PROPERTY PickPlaceDataToPass : ST_PickPlace
GET
PickPlaceDataToPass := _PickPlaceDataToPass;
END_GET
END_PROPERTY

END_FUNCTION_BLOCK

// Machine/EquipmentModules/Functional Layer/FB_Robot_PrePlate
FUNCTION_BLOCK FB_Robot_PrePlate EXTENDS FB_Robot
VAR
    // Sub module definitions here

    Detail_SIM_TON : TON;
END_VAR

VAR

    Plates : ST_Plates;

END_VAR

METHOD CyclicLogic
VAR_INPUT
END_VAR

VAR

END_VAR
IF NOT _InitComplete THEN
    _InitComplete := Initialize();
    RETURN;
END_IF

SUPER^.CyclicLogic();

UI_MessageBox();
END_METHOD

METHOD CyclicLogicSimulation : BOOL
VAR_INPUT
END_VAR
END_METHOD

METHOD ExecuteDetail : BOOL
VAR_INPUT
    StepToRun : UDINT;
END_VAR
ExecuteDetail := FALSE;

CASE Handshake_Step OF
    0:
        Robot.Handshake.OUT.Execute_Step    := TRUE;
        Robot.Handshake.OUT.Execute_StepNum := UDINT_TO_UINT(StepToRun);

        IF Robot.Handshake.IN.Executing_Step = TRUE THEN
            Handshake_Step := 1;
        END_IF

    1:
        IF Robot.Handshake.IN.Executing_Step = FALSE AND Robot.Handshake.IN.StepComplete = TRUE THEN
            Handshake_Step := 2;
        END_IF

    2:
        Robot.Handshake.OUT.Execute_Step    := FALSE;
        Robot.Handshake.OUT.Execute_StepNum := 0;

        IF Robot.Handshake.IN.StepComplete = FALSE THEN
            ExecuteDetail  := TRUE;
            Handshake_Step := 0;
        END_IF

END_CASE
END_METHOD

METHOD PROTECTED ExecuteDetail_SIM : BOOL
VAR_INPUT
    StepToRun : UDINT;
END_VAR
IF WaitSync_Handler(E_WaitSync.PRESS_PREPLATE_SIM_SYNC) THEN
    ExecuteDetail_SIM := TRUE;
END_IF
END_METHOD

METHOD ExecuteStep : BOOL
VAR_INPUT
    Step : ST_CSV_Step;
END_VAR

VAR_INST
    LastExecutionTime  : ULINT; // 64-bit unsigned for F_GetSystemTime
    CurrentTime        : ULINT;
    LastHourCheck      : ULINT;
    ExecutionTime      : ULINT;
    NailPlateTimes     : ARRAY[0..9] OF ULINT; // Buffer for 10 samples
    TotalTime          : REAL; // Use REAL for floating-point calc
    TimeBufferIndex    : INT  := 0;
    TimeSampleCount    : INT  := 0;
    NailPlatesPerMin   : REAL := 0.0; // Plates per minute
    NailPlatesPerHour  : REAL := 0.0; // Plates per hour
    HourAccumulator    : REAL := 0.0;
    ShiftSampleCount   : INT  := 0;
    ShiftNailPlateAvgs : ARRAY[0..7] OF REAL; // 8-hour shift storage
    ShiftHourIndex     : INT := 0;
    BoardNumber        : INT;
END_VAR
ExecuteStep := FALSE;

CASE Step.seqName OF
    E_CommandName.BoardInfo:
        BoardNumber := STRING_TO_INT(Step.Details[1].Datas[2]);
		ExecuteStep := TRUE;
    E_CommandName.NailPlate:
        // Initialize timing on first run
        IF TimeSampleCount = 0 AND TimeBufferIndex = 0 AND ShiftSampleCount = 0 THEN
            LastExecutionTime := F_GetSystemTime();
            LastHourCheck     := LastExecutionTime;
        END_IF

        NailPlateParse(Step, Plates);

        // Clear out array first
        Robot.Clear_DataToSend();

        // First entry is always step type
        Robot.RecipeData_ToSend[0] := E_CommandName.NailPlate;

        Robot.RecipeData_ToSend[1] := UDINT_TO_DINT(Step.DetailCount);
        Robot.RecipeData_ToSend[2] := (Plates.Plates[DetailIndex].PlateNumber + (BoardNumber * 10));
        Robot.RecipeData_ToSend[3] := ExtractNumFromString(Plates.Plates[DetailIndex].PlateGauge);
        Robot.RecipeData_ToSend[4] := REAL_TO_DINT(Plates.Plates[DetailIndex].PlateWidth * 10);
        Robot.RecipeData_ToSend[5] := REAL_TO_DINT(Plates.Plates[DetailIndex].PlateHeight * 10);
        Robot.RecipeData_ToSend[6] := REAL_TO_DINT(Plates.Plates[DetailIndex].PlatePlaceY * 10);
        Robot.RecipeData_ToSend[7] := REAL_TO_DINT(Plates.Plates[DetailIndex].PlatePlaceAngle * 10);

        IF Plates.Plates[DetailIndex].TopOrBottom = 'Top' THEN
            Robot.RecipeData_ToSend[8] := 1;
        ELSIF Plates.Plates[DetailIndex].TopOrBottom = 'Bottom' THEN
            Robot.RecipeData_ToSend[8] := 2;
        ELSE
            Robot.RecipeData_ToSend[8] := 0;
        END_IF

        IF _InSimulation THEN
            IF ExecuteDetail_SIM(Step.seqID) THEN
                DetailIndex := DetailIndex + 1;
                Detail_SIM_TON(IN := FALSE);
            END_IF
        ELSE
            IF ExecuteDetail(Step.seqID) THEN
                CurrentTime   := F_GetSystemTime();
                ExecutionTime := CurrentTime - LastExecutionTime;

                // Convert 100ns units to seconds (100ns * 10,000,000 = 1s)
                NailPlateTimes[TimeBufferIndex] := ExecutionTime;
                TimeBufferIndex                 := TimeBufferIndex + 1;

                IF TimeBufferIndex >= 10 THEN
                    TimeBufferIndex := 0;
                END_IF

                IF TimeSampleCount < 10 THEN
                    TimeSampleCount := TimeSampleCount + 1;
                END_IF

                TotalTime := 0.0;

                FOR i := 0 TO TimeSampleCount - 1 DO
                    TotalTime := TotalTime + ULINT_TO_REAL(NailPlateTimes[i]) / 10000000.0; // Convert to seconds
                END_FOR

                IF TotalTime > 0.0 THEN
                    // Calculate plates per minute (samples per average time in seconds)
                    NailPlatesPerMin := (TimeSampleCount / TotalTime) * 60.0;
                    // Calculate plates per hour
                    NailPlatesPerHour := NailPlatesPerMin * 60.0;
                END_IF

                // Shift-long tracking
                HourAccumulator  := HourAccumulator + 1.0; // Count each plate
                ShiftSampleCount := ShiftSampleCount + 1;

                // Check if an hour has passed (36000000000 100ns units = 1 hour)
                IF (CurrentTime - LastHourCheck) >= 36000000000 THEN
                    IF ShiftSampleCount > 0 THEN
                        // Store hourly rate (plates per hour)
                        ShiftNailPlateAvgs[ShiftHourIndex] := (HourAccumulator * 3600.0) / (ULINT_TO_REAL(CurrentTime - LastHourCheck) / 10000000.0);
                        ShiftHourIndex                     := ShiftHourIndex + 1;
                        HourAccumulator                    := 0.0;
                        ShiftSampleCount                   := 0;
                    END_IF

                    LastHourCheck := CurrentTime;

                    IF ShiftHourIndex >= 8 THEN
                        ShiftHourIndex := 0; // Start new shift
                    END_IF
                END_IF

                LastExecutionTime := CurrentTime;
                DetailIndex       := DetailIndex + 1;
            END_IF
        END_IF

        IF DetailIndex > Step.DetailCount THEN
            DetailIndex := 1;
            ExecuteStep := TRUE;
        END_IF

ELSE
    ExecuteStep := TRUE;

END_CASE
END_METHOD

METHOD HMIControl
VAR_INPUT
END_VAR
END_METHOD

//! @summary Basic module initialization logic
METHOD PROTECTED Initialize : BOOL;
VAR
    i                        : UDINT;
    varInfo                  : __SYSTEM.VAR_INFO;
    AllSubUnitsInitialized   : BOOL := TRUE;
    AllComponentsInitialized : BOOL := TRUE;
END_VAR

//! @description This method is called by <c>CyclicLogic()</c> as required
Initialize := FALSE;

CASE DescendantSequenceState OF
    0:
        RegisterComponent(Robot);

        _LogModeChanges         := FALSE;
        _LogStateChanges        := FALSE;
        DescendantSequenceState := DescendantSequenceState + 10;

    10:
        //Setup Custom modes here

        (*CustomModes(eMode                          :=,
                    sName                          :=,
                    bDisableClearing               :=,
                    bDisableStarting               :=,
                    bDisableSuspended              :=,
                    bDisableStopping               :=,
                    bDisableAborting               :=,
                    bDisableHolding                :=,
                    bDisableHeld                   :=,
                    bDisableUnholding              :=,
                    bDisableSuspending             :=,
                    bDisableUnsuspending           :=,
                    bDisableResetting              :=,
                    bDisableIdle                   :=,
                    bDisableCompleting             :=,
                    bDisableComplete               :=,
                    bEnableUnitModeChangeStopped   :=,
                    bEnableUnitModeChangeIdle      :=,
                    bEnableUnitModeChangeSuspended :=,
                    bEnableUnitModeChangeExecute   :=,
                    bEnableUnitModeChangeAborted   :=,
                    bEnableUnitModeChangeHeld      :=,
                    bEnableUnitModeChangeComplete  :=,
                    bError                         =>,
                    nErrorId                       =>);*)

        DescendantSequenceState := DescendantSequenceState + 10;

    20:
        //Copy Mode names

        FOR i := 1 TO 3 DO
            ModeNames[i] := F_UnitModeToString(UDINT_TO_DINT(i));
        END_FOR

        RegisterExternalController(Controller := fbControlSourceHMI);
        fbControlSourceHMI.CyclicLogic();
        DescendantSequenceState := DescendantSequenceState + 10;

    30:
        //Call the Super

        IF SUPER^.Initialize() THEN
            DescendantSequenceState := DescendantSequenceState + 10;
        END_IF

    40:
        Initialize := TRUE;
END_CASE
END_METHOD

METHOD UI_MessageBox : BOOL
VAR_INPUT
END_VAR

VAR
    result : USINT;
END_VAR
IF Robot.Handshake.IN.ErrorPresent THEN
    CASE Robot.Handshake.IN.MessageNumber OF

        //////////////////////////// PREPLATE ROBOT ERRORS ////////////////////////////
        0:

            // Idle State Should not have an error of 0

            ///////// 1-29 PROCESS ERRORS /////////
        1:
            // PrePlate ERROR_REPEATEDSTEP_R1

            result := RaiseMessageBox(Header   := 'Repeated Step Warning.',
                                      Message1 := 'Robot is trying to repeat last step',
                                      Message3 := 'Choose RETRY to retry check',
                                      Message4 := 'Choose ABORT to reset robot',
                                      Btn3     := 'Retry',
                                      Btn4     := 'Override',
                                      Btn5     := 'Abort',
                                      Severity := TcEventSeverity.Error);

        2:
            // PrePlate ERROR_STEP_NOT_FOUND

            result := RaiseMessageBox(Header   := 'Step Not Found Warning.',
                                      Message1 := 'Robot is trying execute a step that does not exist',
                                      Message2 := 'Choose RETRY to retry check',
                                      Message3 := 'Choose OVERRIDE to override warning',
                                      Message4 := 'Choose ABORT to reset robot',
                                      Btn3     := 'Retry',
                                      Btn4     := 'Override',
                                      Btn5     := 'Abort',
                                      Severity := TcEventSeverity.Error);

        3:
            // PrePlate ERROR_PROCESSING_DATA

            result := RaiseMessageBox(Header   := 'Processing Data Error',
                                      Message1 := 'Check robot log for more information',
                                      Message2 := 'Choose RETRY to retry data processing',
                                      Message3 := 'Choose ABORT to reset robot',
                                      Btn3     := 'RETRY',
                                      Btn5     := 'ABORT',
                                      Severity := TcEventSeverity.Error);

        4:
            // PrePlate ERROR_NORUNUNIT

            result := RaiseMessageBox(Header   := 'IO Device not Connected.',
                                      Message1 := 'Check error log for more details',
                                      Message3 := 'click OK when ready to continue',
                                      Btn5     := 'OK',
                                      Severity := TcEventSeverity.Error);

        5:
            // PrePlate ERROR_NO_DATA_FILE

            result := RaiseMessageBox(Header   := 'No Data File Found.',
                                      Message1 := 'Resend data to robot and choose RETRY',
                                      Message3 := 'Choose ABORT to start recovery process',
                                      Btn3     := 'RETRY',
                                      Btn5     := 'ABORT',
                                      Severity := TcEventSeverity.Error);

        6:
            // PrePlate ERROR_ABORT

            result := RaiseMessageBox(Header   := 'Abort Error',
                                      Message1 := 'Aborting',
                                      Message3 := 'Select ABORT to continue.',
                                      Btn3     := 'ABORT',
                                      Severity := TcEventSeverity.Error);

        10:
            // Press Error ERROR_ABORT (Left magnet handoff not extending)

            result := RaiseMessageBox(Header   := 'Left magnet handoff not extending',
                                      Message1 := 'Make sure air on and extend sensor is connected correctly ',
                                      Message3 := 'System will continue when extend signal is triggered',
                                      Btn3     := 'OVERRIDE',
                                      Severity := TcEventSeverity.Info);

        11:
            // Press Error ERROR_ABORT (Right magnet handoff not extending)

            result := RaiseMessageBox(Header   := 'Right magnet handoff not extending',
                                      Message1 := 'Make sure air on and extend sensor is connected correctly ',
                                      Message3 := 'System will continue when extend signal is triggered',
                                      Btn3     := 'OVERRIDE',
                                      Severity := TcEventSeverity.Info);

        30:
            // PrePlate Error ERROR_UNKNOWNERROR_R1

            result := RaiseMessageBox(Header   := 'Unknown Robot Error',
                                      Message1 := 'Check the pendant for additional information.',
                                      Message3 := 'Press OK to continue.',
                                      Btn5     := 'OK',
                                      Severity := TcEventSeverity.Error);

        31:
            // PrePlate ERROR_PLATEDROPPED_R1

            result := RaiseMessageBox(Header   := 'PrePlate Robot Dropped Plate.',
                                      Message1 := 'Robot no longer holding plate.',
                                      Message3 := 'Choose ABORT to reset robot',
                                      Btn2     := 'Discard',
                                      Btn3     := 'Re-Pick',
                                      Btn4     := 'Override',
                                      Btn5     := 'Abort',
                                      Severity := TcEventSeverity.Error);

        32:
            // PrePlate ERROR_TWO_PLATES_DROPPED

            result := RaiseMessageBox(Header   := 'PrePlate Robot Dropped Plate Twice.',
                                      Message1 := 'Check End Of Arm Tool',
                                      Message3 := 'Choose OVERRIDE if nothing wrong',
                                      Message4 := 'Choose ABORT to reset robot',
                                      Btn2     := 'Discard',
                                      Btn3     := 'Re-Pick',
                                      Btn4     := 'Override',
                                      Btn5     := 'Abort',
                                      Severity := TcEventSeverity.Error);

        33:
            // Press ERROR_NO_MORE_MAGS

            // This one includes dynamic text for plate size

            // We'll place that dynamic content in one message for clarity

            result := RaiseMessageBox(Header   := 'No more magazines.',
                                      Message1 := CONCAT('Plate size = ', Plates.Plates[DetailIndex].PlateDimensions),
                                      Message2 := CONCAT('Plate gauge = ', Plates.Plates[DetailIndex].PlateGauge),
                                      Message3 := 'click OK when magazines are filled',
                                      Btn3     := 'Skip',
                                      Btn5     := 'OK',
                                      Severity := TcEventSeverity.Error);

        34:
            // PrePlate ERROR_EOAT_EXT_FAILURE

            result := RaiseMessageBox(Header   := 'EOAT Failed to Extend.',
                                      Message1 := 'Check EOAT for any blockage',
                                      Message2 := 'Choose DISABLE to disable check',
                                      Message3 := 'Choose RETRY to retry check',
                                      Message4 := 'Choose OVERRIDE to override warning',
                                      Message5 := 'Choose ABORT to reset robot',
                                      Btn2     := 'Disable',
                                      Btn3     := 'Retry',
                                      Btn4     := 'Override',
                                      Btn5     := 'Abort',
                                      Severity := TcEventSeverity.Error);

        35:
            // PrePlate ERROR_PLATE_NOT_FOUND

            result := RaiseMessageBox(Header   := 'Specified Plate does not Exist.',
                                      Message1 := 'Check data',
                                      Message2 := 'Choose RETRY to retry check',
                                      Message3 := 'Choose OVERRIDE to override warning',
                                      Message4 := 'Choose ABORT to reset robot',
                                      Btn3     := 'Retry',
                                      Btn4     := 'Override',
                                      Btn5     := 'Abort',
                                      Severity := TcEventSeverity.Error);

        36:
            // PrePlate ERROR_PLACE_OUT_OF_REACH

            result := RaiseMessageBox(Header   := 'Robot Out of Reach',
                                      Message1 := 'Check data',
                                      Message3 := 'Choose DISCARD to discard plate and move on to next one.',
                                      Btn3     := 'DISCARD',
                                      Btn5     := 'RECOVER',
                                      Severity := TcEventSeverity.Error);

        37:
            // PrePlate ERROR_UNRECOGNIZED_WORLD_ZONE

            result := RaiseMessageBox(Header   := 'Robot Unrecognized Position.',
                                      Message1 := 'Jog Robot to safe position and retry move home',
                                      Btn5     := 'RETRY',
                                      Severity := TcEventSeverity.Error);

        38:
            // PrePlate ERROR_PRESS_TASK_STOPPED

            result := RaiseMessageBox(Header   := 'Press Task Stopped.',
                                      Message1 := 'Make sure all tasks are enabled on the robot.',
                                      Btn5     := 'Retry',
                                      Severity := TcEventSeverity.Error);

        40:
            // PrePlate ERROR_NO_HANDSHAKE_ROBOT

            result := RaiseMessageBox(Header   := 'Robot - Waiting to Handshake',
                                      Message1 := 'The PLC and robot may be out of sync',
                                      Btn5     := 'Retry',
                                      Severity := TcEventSeverity.Error);

        41:
            // PrePlate ERROR_BAD_BOARD_DATA

            result := RaiseMessageBox(Header   := 'Bad Board Data',
                                      Message1 := 'Preplate CSV board data has boards that are too long/short/thick to be ran',
                                      Message3 := 'Check files and upload new files when fixed',
                                      Severity := TcEventSeverity.Error);

        42:
            // PrePlate ERROR_BAD_NAIL_DATA

            result := RaiseMessageBox(Header   := 'Bad Nail Plate Data',
                                      Message1 := 'Preplate CSV nail plate data has incorrect plate sizes',
                                      Message3 := 'Check files and upload new files when fixed',
                                      Severity := TcEventSeverity.Error);

        43:
            // PrePlate ERROR_FAILED_TO_PLACE

            result := RaiseMessageBox(Header   := 'PP Robot Failed to Place Nail Plate',
                                      Message1 := 'PrePlate robot still holding a nail plate after attempting to place it',
                                      Message3 := 'Select RETRY to have robot attempt to place nail plate again',
                                      Btn3     := 'Retry',
                                      Severity := TcEventSeverity.Error);

        44:
            // PrePlate ERROR_MAG_IN_DIS_RACK

            result := RaiseMessageBox(Header   := 'Only Available Magazine is in a Disabled Rack',
                                      Message1 := 'Re-Enable Rack',
                                      Message3 := 'Choose RETRY to attempt Finding Valid Mgazine',
                                      Btn5     := 'Retry',
                                      Severity := TcEventSeverity.Error);

        45:
            // PrePlate error nail plate skipped

            // Also includes dynamic text for plate size

            result := RaiseMessageBox(Header   := 'Nail plate Skipped',
                                      Message1 := 'Nail plate not available',
                                      Message3 := CONCAT('Nail plate size: ', Plates.Plates[DetailIndex].PlateDimensions),
                                      Btn5     := 'OK',
                                      Severity := TcEventSeverity.Error);

        50:
            result := RaiseMessageBox(Header   := 'Robot Read Bad Board Data',
                                      Message1 := 'Preplate CSV board data has boards that are too long/short/thick to be ran',
                                      Message3 := 'Check files and upload new files when fixed',
                                      Severity := TcEventSeverity.Error);

        60:
            // PrePlate MESSAGE_ATSERVICE_R1

            result := RaiseMessageBox(Header   := 'Robot at Service Position.',
                                      Message1 := 'Choose DONE when ready to return robot to home',
                                      Btn5     := 'DONE',
                                      Severity := TcEventSeverity.Error);

        61:
            // PrePlate MESSAGE_PLATE_ON_MAGNET

            result := RaiseMessageBox(Header   := 'Plate(s) Likely Left on Handoff Magnet(s)',
                                      Message1 := 'Choose REMOVE to allow robot to remove plate',
                                      Message3 := 'Choose CONTINUE if plate are removed manually',
                                      Btn4     := 'REMOVE',
                                      Btn5     := 'CONTINUE',
                                      Severity := TcEventSeverity.Error);

        62:
            // PrePlate MESSAGE_GET_RECOVERY

            result := RaiseMessageBox(Header   := 'Choose Restart Option',
                                      Message1 := 'Choose FULL ABORT to clear out truss',
                                      Message2 := 'Choose SKIP BOARD to skip to next board in recipe',
                                      Message3 := 'Choose RESTART BOARD to remove board and restart plating',
                                      Message4 := 'Choose SKIP PLATE to discard plate and restart from next plate',
                                      Message5 := 'Choose RECOVER STEP to remove board and restart form specified board',
                                      Btn1     := 'FULL ABORT',
                                      Btn2     := 'SKIP BOARD',
                                      Btn3     := 'RESTART BOARD',
                                      Btn4     := 'SKIP PLATE',
                                      Btn5     := 'RECOVER STEP',
                                      Severity := TcEventSeverity.Error);

        63:
            // PrePlate MESSAGE_BOARD_RESTART

            // UI_MessageBoxes.UI_MessageBox[2].Recover.Visible := TRUE;

            // UI_MessageBoxes.UI_MessageBox[2].Recover.BoardData := gBoardData;

            result := RaiseMessageBox(Header   := 'Select Board to Restart',
                                      Message1 := 'Select a board to start on',
                                      Message3 := 'Select OK when system is ready to continue',
                                      Btn1     := 'Cancel',
                                      Btn5     := 'OK',
                                      Severity := TcEventSeverity.Error);

        64:
            // PrePlate MESSAGE_PLATE_RESTART

            // UI_MessageBoxes.UI_MessageBox[2].NumEntry.Visible := TRUE;

            result := RaiseMessageBox(Header   := 'Specify Plate to Restart',
                                      Message1 := 'Select a plate to start on',
                                      Btn5     := 'OK',
                                      Severity := TcEventSeverity.Error);

        65:
            // PrePlate MESSAGE_CONFIRM_SKIP

            result := RaiseMessageBox(Header   := 'Confirm Skip Current Step',
                                      Message1 := 'Are you sure you want to skip current step?',
                                      Btn1     := 'GO BACK',
                                      Btn5     := 'CONFIRM',
                                      Severity := TcEventSeverity.Error);

        66:
            // PrePlate MESSAGE_CONFIRM_RETRY

            result := RaiseMessageBox(Header   := 'Confirm Retry Current Step',
                                      Message1 := 'Are you sure you want to retry current step?',
                                      Btn1     := 'GO BACK',
                                      Btn5     := 'CONFIRM',
                                      Severity := TcEventSeverity.Error);

        67:
            // PrePlate MESSAGE_CONFIRM_ABORT

            result := RaiseMessageBox(Header   := 'Confirm Abort Current Truss',
                                      Message1 := 'Are you sure you want to abort current truss?',
                                      Btn1     := 'GO BACK',
                                      Btn5     := 'CONFIRM',
                                      Severity := TcEventSeverity.Error);

        68:
            // PrePlate MESSAGE_CONFIRM_RECOVER

            result := RaiseMessageBox(Header   := 'Confirm Recover Current Truss',
                                      Message1 := 'Are you sure you want to recover current truss?',
                                      Btn1     := 'GO BACK',
                                      Btn5     := 'CONFIRM',
                                      Severity := TcEventSeverity.Error);

        69:
            // PrePlate MESSAGE_CONFIRM_SKIP_PLATE

            result := RaiseMessageBox(Header   := 'Confirm Skip Current Plate',
                                      Message1 := 'Are you sure you want to skip current plate?',
                                      Btn1     := 'GO BACK',
                                      Btn5     := 'CONFIRM',
                                      Severity := TcEventSeverity.Error);

        70:
            // PrePlate Failed to remove nail plate

            result := RaiseMessageBox(Header   := 'Robot failed to clear plate from handoff',
                                      Message1 := 'Remove plate manually.',
                                      Message2 := 'Choose OK to continue.',
                                      Btn5     := 'OK',
                                      Severity := TcEventSeverity.Error);

    ELSE
        // Not Valid Message Number

        // The original code appends the ErrorNumber integer to the message.

        // We'll keep the same logic, but we can store it as a separate or inline string.

        // For demonstration, we directly pass in the integer, though we normally would do

        // a conversion. We'll just label it as an unknown message.

        result := RaiseMessageBox(Header   := 'Not Valid Message Number',
                                  Message1 := CONCAT('UIMessageBox was sent message number: ', UINT_TO_STRING(Robot.Handshake.IN.MessageNumber)),
                                  Message3 := 'Contact Support to update message number.',
                                  Btn1     := 'EXIT MSG',
                                  Severity := TcEventSeverity.Error);
    END_CASE;

    IF result <> 0 THEN
        Robot.Handshake.OUT.MessageSolution    := result;
        Robot.Handshake.OUT.MessageAcknowledge := TRUE;
    END_IF
ELSE
    Robot.Handshake.OUT.MessageSolution    := 0;
    Robot.Handshake.OUT.MessageAcknowledge := FALSE;
END_IF;
END_METHOD

END_FUNCTION_BLOCK

// Machine/EquipmentModules/Functional Layer/FB_Robot_Press
FUNCTION_BLOCK FB_Robot_Press EXTENDS FB_Robot

VAR

    Plates : ST_Plates;

END_VAR

METHOD CyclicLogic
VAR_INPUT
END_VAR

VAR

END_VAR
IF NOT _InitComplete THEN
    _InitComplete := Initialize();
    RETURN;
END_IF

SUPER^.CyclicLogic();

UI_MessageBox();
END_METHOD

METHOD CyclicLogicSimulation : BOOL
VAR_INPUT
END_VAR
END_METHOD

METHOD ExecuteDetail : BOOL
VAR_INPUT
    StepToRun : UDINT;
END_VAR
ExecuteDetail := FALSE;

CASE Handshake_Step OF
    0:
        Robot.Handshake.OUT.Execute_Step    := TRUE;
        Robot.Handshake.OUT.Execute_StepNum := UDINT_TO_UINT(StepToRun);

        IF Robot.Handshake.IN.Executing_Step = TRUE THEN
            Handshake_Step := 1;
        END_IF

    1:
        IF Robot.Handshake.IN.Executing_Step = FALSE AND Robot.Handshake.IN.StepComplete = TRUE THEN
            Handshake_Step := 2;
        END_IF

    2:
        Robot.Handshake.OUT.Execute_Step    := FALSE;
        Robot.Handshake.OUT.Execute_StepNum := 0;

        IF Robot.Handshake.IN.StepComplete = FALSE THEN
            ExecuteDetail  := TRUE;
            Handshake_Step := 0;
        END_IF

END_CASE
END_METHOD

METHOD PROTECTED ExecuteDetail_SIM : BOOL
VAR_INPUT
    StepToRun : UDINT;
END_VAR

VAR_INST
    robotWS_State : E_Press_States;
END_VAR
CASE robotWS_State OF
    PRESS_INIT:
        IF WaitSync_Handler(E_WaitSync.PRESS_PREPLATE_SIM_SYNC) THEN
            robotWS_State := ROBOT_PERMISSION_REQUEST;
        END_IF

    ROBOT_PERMISSION_REQUEST:
        IF WaitSync_Handler(E_WaitSync.NAILPLATE_READY_TO_PLACE) THEN
            robotWS_State := ROBOT_PERMISSION_GRANTED_WS;
        END_IF

    ROBOT_PERMISSION_GRANTED_WS:
        IF WaitSync_Handler(E_WaitSync.PRESS_ROBOT_PERMISSION_GRANTED) THEN
            robotWS_State := NP_PLACED_WS;
        END_IF

    NP_PLACED_WS:
        IF WaitSync_Handler(E_WaitSync.NAILPLATE_PLACED) THEN
            robotWS_State := NP_DONE_WS;
        END_IF

    NP_DONE_WS:
        ExecuteDetail_SIM := true;
        robotWS_State     := PRESS_INIT;
END_CASE
END_METHOD

METHOD ExecuteStep : BOOL
VAR_INPUT
    Step : ST_CSV_Step;
END_VAR

VAR_INST
    LastExecutionTime  : ULINT; // 64-bit unsigned for F_GetSystemTime
    CurrentTime        : ULINT;
    LastHourCheck      : ULINT;
    ExecutionTime      : ULINT;
    NailPlateTimes     : ARRAY[0..9] OF ULINT; // Buffer for 10 samples
    TotalTime          : REAL; // Use REAL for floating-point calc
    TimeBufferIndex    : INT  := 0;
    TimeSampleCount    : INT  := 0;
    NailPlatesPerMin   : REAL := 0.0; // Plates per minute
    NailPlatesPerHour  : REAL := 0.0; // Plates per hour
    HourAccumulator    : REAL := 0.0;
    ShiftSampleCount   : INT  := 0;
    ShiftNailPlateAvgs : ARRAY[0..7] OF REAL; // 8-hour shift storage
    ShiftHourIndex     : INT := 0;
    BoardNumber        : INT;
END_VAR
ExecuteStep := FALSE;

CASE Step.seqName OF
    E_CommandName.BoardInfo:
        BoardNumber := STRING_TO_INT(Step.Details[1].Datas[2]);
		ExecuteStep := TRUE;
    E_CommandName.NailPlate:

        NailPlateParse(Step, Plates);

        // clear out array first
        Robot.Clear_DataToSend();

        // first entry is always step type
        Robot.RecipeData_ToSend[0] := E_CommandName.NailPlate;

        Robot.RecipeData_ToSend[1] := UDINT_TO_DINT(Step.DetailCount);

        Robot.RecipeData_ToSend[2] := (Plates.Plates[DetailIndex].PlateNumber + (BoardNumber * 10));

        Robot.RecipeData_ToSend[3] := ExtractNumFromString(Plates.Plates[DetailIndex].PlateGauge);

        Robot.RecipeData_ToSend[4] := REAL_TO_DINT(Plates.Plates[DetailIndex].PlateWidth * 10);

        Robot.RecipeData_ToSend[5] := REAL_TO_DINT(Plates.Plates[DetailIndex].PlateHeight * 10);

        Robot.RecipeData_ToSend[6] := REAL_TO_DINT(Plates.Plates[DetailIndex].PlatePlaceY * 10);

        Robot.RecipeData_ToSend[7] := REAL_TO_DINT(Plates.Plates[DetailIndex].PlatePlaceAngle * 10);

        IF Plates.Plates[DetailIndex].TopOrBottom = 'Top' THEN
            Robot.RecipeData_ToSend[8] := 1;
        ELSIF Plates.Plates[DetailIndex].TopOrBottom = 'Bottom' THEN
            Robot.RecipeData_ToSend[8] := 2;
        ELSE
            Robot.RecipeData_ToSend[8] := 0;
        END_IF

        IF _InSimulation THEN
            IF ExecuteDetail_SIM(Step.seqID) THEN
                DetailIndex := DetailIndex + 1;
				                CurrentTime   := F_GetSystemTime();
                ExecutionTime := CurrentTime - LastExecutionTime;

                // Convert 100ns units to seconds (100ns * 10,000,000 = 1s)
                NailPlateTimes[TimeBufferIndex] := ExecutionTime;
                TimeBufferIndex                 := TimeBufferIndex + 1;

                IF TimeBufferIndex >= 10 THEN
                    TimeBufferIndex := 0;
                END_IF

                IF TimeSampleCount < 10 THEN
                    TimeSampleCount := TimeSampleCount + 1;
                END_IF

                TotalTime := 0.0;

                FOR i := 0 TO TimeSampleCount - 1 DO
                    TotalTime := TotalTime + ULINT_TO_REAL(NailPlateTimes[i]) / 10000000.0; // Convert to seconds
                END_FOR

                IF TotalTime > 0.0 THEN
                    // Calculate plates per minute (samples per average time in seconds)
                    NailPlatesPerMin := (TimeSampleCount / TotalTime) * 60.0;
                    // Calculate plates per hour
                    NailPlatesPerHour := NailPlatesPerMin * 60.0;
                END_IF

                // Shift-long tracking
                HourAccumulator  := HourAccumulator + 1.0; // Count each plate
                ShiftSampleCount := ShiftSampleCount + 1;

                // Check if an hour has passed (36000000000 100ns units = 1 hour)
                IF (CurrentTime - LastHourCheck) >= 36000000000 THEN
                    IF ShiftSampleCount > 0 THEN
                        // Store hourly rate (plates per hour)
                        ShiftNailPlateAvgs[ShiftHourIndex] := (HourAccumulator * 3600.0) / (ULINT_TO_REAL(CurrentTime - LastHourCheck) / 10000000.0);
                        ShiftHourIndex                     := ShiftHourIndex + 1;
                        HourAccumulator                    := 0.0;
                        ShiftSampleCount                   := 0;
                    END_IF

                    LastHourCheck := CurrentTime;

                    IF ShiftHourIndex >= 8 THEN
                        ShiftHourIndex := 0; // Start new shift
                    END_IF
                END_IF

                LastExecutionTime := CurrentTime;


            END_IF
        ELSE
            IF ExecuteDetail(Step.seqID) THEN
                CurrentTime   := F_GetSystemTime();
                ExecutionTime := CurrentTime - LastExecutionTime;

                // Convert 100ns units to seconds (100ns * 10,000,000 = 1s)
                NailPlateTimes[TimeBufferIndex] := ExecutionTime;
                TimeBufferIndex                 := TimeBufferIndex + 1;

                IF TimeBufferIndex >= 10 THEN
                    TimeBufferIndex := 0;
                END_IF

                IF TimeSampleCount < 10 THEN
                    TimeSampleCount := TimeSampleCount + 1;
                END_IF

                TotalTime := 0.0;

                FOR i := 0 TO TimeSampleCount - 1 DO
                    TotalTime := TotalTime + ULINT_TO_REAL(NailPlateTimes[i]) / 10000000.0; // Convert to seconds
                END_FOR

                IF TotalTime > 0.0 THEN
                    // Calculate plates per minute (samples per average time in seconds)
                    NailPlatesPerMin := (TimeSampleCount / TotalTime) * 60.0;
                    // Calculate plates per hour
                    NailPlatesPerHour := NailPlatesPerMin * 60.0;
                END_IF

                // Shift-long tracking
                HourAccumulator  := HourAccumulator + 1.0; // Count each plate
                ShiftSampleCount := ShiftSampleCount + 1;

                // Check if an hour has passed (36000000000 100ns units = 1 hour)
                IF (CurrentTime - LastHourCheck) >= 36000000000 THEN
                    IF ShiftSampleCount > 0 THEN
                        // Store hourly rate (plates per hour)
                        ShiftNailPlateAvgs[ShiftHourIndex] := (HourAccumulator * 3600.0) / (ULINT_TO_REAL(CurrentTime - LastHourCheck) / 10000000.0);
                        ShiftHourIndex                     := ShiftHourIndex + 1;
                        HourAccumulator                    := 0.0;
                        ShiftSampleCount                   := 0;
                    END_IF

                    LastHourCheck := CurrentTime;

                    IF ShiftHourIndex >= 8 THEN
                        ShiftHourIndex := 0; // Start new shift
                    END_IF
                END_IF

                LastExecutionTime := CurrentTime;

                DetailIndex := DetailIndex + 1;
            END_IF
        END_IF

        IF DetailIndex > Step.DetailCount THEN
            DetailIndex := 1;
            ExecuteStep := TRUE;
        END_IF

ELSE
    ExecuteStep := TRUE;

END_CASE
END_METHOD

METHOD HMIControl
VAR_INPUT
END_VAR
END_METHOD

//! @summary Basic module initialization logic
METHOD PROTECTED Initialize : BOOL;
VAR
    i                        : UDINT;
    varInfo                  : __SYSTEM.VAR_INFO;
    AllSubUnitsInitialized   : BOOL := TRUE;
    AllComponentsInitialized : BOOL := TRUE;
END_VAR

//! @description This method is called by <c>CyclicLogic()</c> as required
Initialize := FALSE;

CASE DescendantSequenceState OF
    0:
        RegisterComponent(Robot);

        _LogModeChanges         := FALSE;
        _LogStateChanges        := FALSE;
        DescendantSequenceState := DescendantSequenceState + 10;

    10:
        //Setup Custom modes here

        (*CustomModes(eMode                          :=,
                    sName                          :=,
                    bDisableClearing               :=,
                    bDisableStarting               :=,
                    bDisableSuspended              :=,
                    bDisableStopping               :=,
                    bDisableAborting               :=,
                    bDisableHolding                :=,
                    bDisableHeld                   :=,
                    bDisableUnholding              :=,
                    bDisableSuspending             :=,
                    bDisableUnsuspending           :=,
                    bDisableResetting              :=,
                    bDisableIdle                   :=,
                    bDisableCompleting             :=,
                    bDisableComplete               :=,
                    bEnableUnitModeChangeStopped   :=,
                    bEnableUnitModeChangeIdle      :=,
                    bEnableUnitModeChangeSuspended :=,
                    bEnableUnitModeChangeExecute   :=,
                    bEnableUnitModeChangeAborted   :=,
                    bEnableUnitModeChangeHeld      :=,
                    bEnableUnitModeChangeComplete  :=,
                    bError                         =>,
                    nErrorId                       =>);*)

        DescendantSequenceState := DescendantSequenceState + 10;

    20:
        //Copy Mode names

        FOR i := 1 TO 3 DO
            ModeNames[i] := F_UnitModeToString(UDINT_TO_DINT(i));
        END_FOR

        RegisterExternalController(Controller := fbControlSourceHMI);
        fbControlSourceHMI.CyclicLogic();
        DescendantSequenceState := DescendantSequenceState + 10;

    30:
        //Call the Super

        IF SUPER^.Initialize() THEN
            DescendantSequenceState := DescendantSequenceState + 10;
        END_IF

    40:
        Initialize := TRUE;
END_CASE
END_METHOD

METHOD UI_MessageBox : BOOL
VAR_INPUT
END_VAR

VAR
    result : USINT;
END_VAR
IF Robot.Handshake.IN.ErrorPresent THEN
    CASE Robot.Handshake.IN.MessageNumber OF

        //////////////////////////// Press ROBOT ERRORS ////////////////////////////
        0:

            // Idle State - Should not have an error of 0

            ///////// 1-29 PROCESS ERRORS /////////
        1:
            // Press ERROR_REPEATEDSTEP_R1 (Already converted)
            result := RaiseMessageBox(Header   := 'Repeated Step Warning.',
                                      Message1 := 'Robot is trying to repeat last step',
                                      Message2 := 'Choose RETRY to retry check',
                                      Message3 := 'Choose ABORT to reset robot',
                                      Btn3     := 'Retry',
                                      Btn4     := 'Override',
                                      Btn5     := 'Abort',
                                      Severity := TcEventSeverity.Error);

        2:
            // Press ERROR_STEP_NOT_FOUND
            result := RaiseMessageBox(Header   := 'Step Not Found Warning.',
                                      Message1 := 'Robot is trying execute a step that does not exist',
                                      Message2 := 'Choose RETRY to retry check',
                                      Message3 := 'Choose OVERRIDE to override warning',
                                      Message4 := 'Choose ABORT to reset robot',
                                      Btn3     := 'Retry',
                                      Btn4     := 'Override',
                                      Btn5     := 'Abort',
                                      Severity := TcEventSeverity.Error);

        3:
            // Press ERROR_PROCESSING_DATA
            result := RaiseMessageBox(Header   := 'Processing Data Error',
                                      Message1 := 'Check robot log for more information',
                                      Message2 := 'Choose RETRY to retry data processing',
                                      Message3 := 'Choose ABORT to reset robot',
                                      Btn3     := 'RETRY',
                                      Btn5     := 'Abort',
                                      Severity := TcEventSeverity.Error);

        4:
            // Press ERROR_NORUNUNIT
            result := RaiseMessageBox(Header   := 'IO Device not Connected.',
                                      Message1 := 'Check error log for more details',
                                      Message3 := 'click OK when ready to continue',
                                      Btn5     := 'OK',
                                      Severity := TcEventSeverity.Error);

        5:
            // Press ERROR_NO_DATA_FILE
            result := RaiseMessageBox(Header   := 'No Data File Found.',
                                      Message1 := 'Resend data to robot and choose RETRY',
                                      Message3 := 'Choose ABORT to start recovery process',
                                      Btn3     := 'RETRY',
                                      Btn5     := 'ABORT',
                                      Severity := TcEventSeverity.Error);

        6:
            // Press ERROR_ABORT
            result := RaiseMessageBox(Header   := 'Abort Error',
                                      Message1 := 'Aborting',
                                      Message3 := 'Select ABORT to continue.',
                                      Btn3     := 'ABORT',
                                      Severity := TcEventSeverity.Error);

        10:
            // Press Error ERROR_ABORT
            result := RaiseMessageBox(Header   := 'Left magnet handoff not retracting',
                                      Message1 := 'Make sure air on and retract sensor is connected correctly ',
                                      Message3 := 'System will continue when retract signal is triggered',
                                      Btn3     := 'OVERRIDE',
                                      Severity := TcEventSeverity.Info);

        11:
            // Press Error ERROR_ABORT
            result := RaiseMessageBox(Header   := 'Right magnet handoff not retracting',
                                      Message1 := 'Make sure air on and retract sensor is connected correctly ',
                                      Message3 := 'System will continue when retract signal is triggered',
                                      Btn3     := 'OVERRIDE',
                                      Severity := TcEventSeverity.Info);

        30:
            // Press Error ERROR_UNKNOWNERROR_R1
            result := RaiseMessageBox(Header   := 'Unknown Robot Error',
                                      Message1 := 'Check the pendant for additional information.',
                                      Message3 := 'Press OK to continue.',
                                      Btn5     := 'OK',
                                      Severity := TcEventSeverity.Error);

        31:
            // Press ERROR_PLATEDROPPED_R1
            result := RaiseMessageBox(Header   := 'Robot Dropped Plate.',
                                      Message1 := 'Robot no longer holding plate.',
                                      Btn4     := 'Override',
                                      Severity := TcEventSeverity.Info);

        32:
            // Press ERROR_TWO_PLATES_DROPPED
            result := RaiseMessageBox(Header   := 'Robot Dropped Plate Twice.',
                                      Message1 := 'Check End Of Arm Tool',
                                      Message2 := 'Choose OVERRIDE if nothing wrong',
                                      Message3 := 'Choose ABORT to reset robot',
                                      Btn2     := 'Discard',
                                      Btn4     := 'Override',
                                      Btn5     := 'Abort',
                                      Severity := TcEventSeverity.Info);

        33:
            // Press ERROR_NO_MORE_MAGS

            // This one includes dynamic text for plate size

            // We'll place that dynamic content in one message for clarity
            result := RaiseMessageBox(Header   := 'No more magazines.',
                                      Message1 := CONCAT('Plate size = ', Plates.Plates[DetailIndex].PlateDimensions),
                                      Message3 := 'click OK when magazines are filled',
                                      Btn5     := 'OK',
                                      Severity := TcEventSeverity.Error);

        34:
            // Press ERROR_EOAT_EXT_FAILURE
            result := RaiseMessageBox(Header   := 'EOAT Failed to Extend.',
                                      Message1 := 'Check EOAT for any blockage',
                                      Message2 := 'Choose DISABLE to disable check',
                                      Message3 := 'Choose RETRY to retry check',
                                      Message4 := 'Choose OVERRIDE to override warning',
                                      Message5 := 'Choose ABORT to reset robot',
                                      Btn2     := 'Disable',
                                      Btn3     := 'Retry',
                                      Btn4     := 'Override',
                                      Btn5     := 'Abort',
                                      Severity := TcEventSeverity.Error);

        35:
            // Press ERROR_PLATE_NOT_FOUND
            result := RaiseMessageBox(Header   := 'Specified Plate does not Exist.',
                                      Message1 := 'Check data',
                                      Message2 := 'Choose RETRY to retry check',
                                      Message3 := 'Choose OVERRIDE to override warning',
                                      Message4 := 'Choose ABORT to reset robot',
                                      Btn3     := 'Retry',
                                      Btn4     := 'Override',
                                      Btn5     := 'Abort',
                                      Severity := TcEventSeverity.Error);

        36:
            // Press ERROR_PLACE_OUT_OF_REACH
            result := RaiseMessageBox(Header   := 'Robot Out of Reach',
                                      Message1 := 'Check data',
                                      Message2 := 'Remove the plate from the Press robot tool.',
                                      Message3 := 'After plate is removed hit SKIP to move on.',
                                      Message4 := 'Choose ABORT to reset robot',
                                      Btn3     := 'SKIP',
                                      Btn5     := 'RECOVER',
                                      Severity := TcEventSeverity.Error);

        37:
            // Press ERROR_UNRECOGNIZED_WORLD_ZONE
            result := RaiseMessageBox(Header   := 'Robot Unrecognized Position.',
                                      Message1 := 'Jog Robot to safe position and retry move home',
                                      Btn5     := 'RETRY',
                                      Severity := TcEventSeverity.Error);

        38:
            // Press ERROR_PLATENOTDROPPED_R1
            result := RaiseMessageBox(Header   := 'Robot Didnt Drop Plate.',
                                      Message1 := 'Check EOAT and press for plates.',
                                      Message2 := 'Choose OVERRIDE to override sensor.',
                                      Message3 := 'Check RETRY to retry plate placement.',
                                      Btn4     := 'Override',
                                      Btn5     := 'Retry',
                                      Severity := TcEventSeverity.Error);

        40:
            // Press ERROR_NO_HANDSHAKE_ROBOT
            result := RaiseMessageBox(Header   := 'Robot - Waiting to Handshake',
                                      Message1 := 'The PLC and robot may be out of sync',
                                      Btn5     := 'Retry',
                                      Severity := TcEventSeverity.Error);

        41:
            // Press ERROR_BAD_BOARD_DATA
            result := RaiseMessageBox(Header   := 'Bad Board Data',
                                      Message1 := 'Preplate CSV board data has boards that are too long/short/thick to be ran',
                                      Message3 := 'Check files and upload new files when fixed',
                                      Severity := TcEventSeverity.Error);

        42:
            // Press ERROR_BAD_NAIL_DATA
            result := RaiseMessageBox(Header   := 'Bad Nail Plate Data',
                                      Message1 := 'Preplate CSV nail plate data has incorrect plate positions',
                                      Message3 := 'Check files and upload new files when fixed',
                                      Severity := TcEventSeverity.Error);

        43:
            // Press ERROR_PLATE_OFFSET_TIMEOUT
            result := RaiseMessageBox(Header   := 'Timeout updating plate offsets with PLC',
                                      Message1 := 'Timeout updating plate offsets with PLC',
                                      Btn3     := 'Retry',
                                      Btn4     := 'Override',
                                      Severity := TcEventSeverity.Error);

        44:
            // PrePlate ERROR_MAG_IN_DIS_RACK

            // Also sets gTrigger_Bool[8]
            result := RaiseMessageBox(Header   := 'Only Available Magazine is in a Disabled Rack',
                                      Message1 := 'Re-Enable Rack',
                                      Message3 := 'Choose RETRY to attempt Finding Valid Mgazine',
                                      Btn5     := 'Retry',
                                      Severity := TcEventSeverity.Error);

        45:
            // PrePlate error nail plate skipped

            // Also includes dynamic text for plate size
            result := RaiseMessageBox(Header   := 'Nail plate Skipped',
                                      Message1 := 'Nail plate not available',
                                      Message3 := CONCAT('Nail plate size: ', Plates.Plates[DetailIndex].PlateDimensions),
                                      Btn5     := 'OK',
                                      Severity := TcEventSeverity.Error);

        50:
            // Press ERROR: Robot Read Bad Board Data
            result := RaiseMessageBox(Header   := 'Robot Read Bad Board Data',
                                      Message1 := 'Preplate CSV board data has boards that are too long/short/thick to be ran',
                                      Message3 := 'Check files and upload new files when fixed',
                                      Severity := TcEventSeverity.Error);

        60:
            // Press MESSAGE_ATSERVICE_R1
            result := RaiseMessageBox(Header   := 'Robot at Service Position.',
                                      Message1 := 'Choose DONE when ready to return robot to home',
                                      Btn5     := 'DONE',
                                      Severity := TcEventSeverity.Error);

        61:
            // Press MESSAGE_PLATE_ON_EOAT
            result := RaiseMessageBox(Header   := 'Plate left on press EOAT.',
                                      Message1 := 'Remove plate and choose OK to continue',
                                      Btn5     := 'OK',
                                      Severity := TcEventSeverity.Error);

        62:
            // Press MESSAGE_GET_RECOVERY
            result := RaiseMessageBox(Header   := 'Choose Restart Option',
                                      Message1 := 'Choose FULL ABORT to clear out truss',
                                      Message2 := 'Choose SKIP BOARD to skip to next board in recipe',
                                      Message3 := 'Choose RESTART BOARD to remove board and restart plating',
                                      Message4 := 'Choose SKIP PLATE to discard plate and restart from next plate',
                                      Message5 := 'Choose RECOVER FROM STEP to remove board and restart form specified board',
                                      Btn1     := 'FULL ABORT',
                                      Btn2     := 'SKIP BOARD',
                                      Btn3     := 'RESTART BOARD',
                                      Btn4     := 'SKIP PLATE',
                                      Btn5     := 'RECOVER FROM STEP',
                                      Severity := TcEventSeverity.Error);

        63:
            // Press MESSAGE_BOARD_RESTART

            // UI_MessageBoxes.UI_MessageBox[1].Recover.Visible := TRUE;

            // UI_MessageBoxes.UI_MessageBox[1].Recover.BoardData := gBoardData;
            result := RaiseMessageBox(Header   := 'Select Board to Restart',
                                      Message1 := 'Select a board to start on',
                                      Message3 := 'Select OK when system is ready to continue',
                                      Btn1     := 'Cancel',
                                      Btn5     := 'OK',
                                      Severity := TcEventSeverity.Error);

        64:
            // Press MESSAGE_PLATE_RESTART

            // UI_MessageBoxes.UI_MessageBox[1].NumEntry.Visible := TRUE;
            result := RaiseMessageBox(Header   := 'Specify Plate to Restart',
                                      Message1 := 'Select a plate to start on',
                                      Btn5     := 'OK',
                                      Severity := TcEventSeverity.Error);

        65:
            // Press MESSAGE_CONFIRM_SKIP
            result := RaiseMessageBox(Header   := 'Confirm Skip Current Step',
                                      Message1 := 'Are you sure you want to skip current step?',
                                      Btn1     := 'GO BACK',
                                      Btn5     := 'CONFIRM',
                                      Severity := TcEventSeverity.Error);

        66:
            // Press MESSAGE_CONFIRM_RETRY
            result := RaiseMessageBox(Header   := 'Confirm Retry Current Step',
                                      Message1 := 'Are you sure you want to retry current step?',
                                      Btn1     := 'GO BACK',
                                      Btn5     := 'CONFIRM',
                                      Severity := TcEventSeverity.Error);

        67:
            // Press MESSAGE_CONFIRM_ABORT
            result := RaiseMessageBox(Header   := 'Confirm Abort Current Truss',
                                      Message1 := 'Are you sure you want to abort current truss?',
                                      Btn1     := 'GO BACK',
                                      Btn5     := 'CONFIRM',
                                      Severity := TcEventSeverity.Error);

        68:
            // Press MESSAGE_CONFIRM_RECOVER
            result := RaiseMessageBox(Header   := 'Confirm Recover Current Truss',
                                      Message1 := 'Are you sure you want to recover current truss?',
                                      Btn1     := 'GO BACK',
                                      Btn5     := 'CONFIRM',
                                      Severity := TcEventSeverity.Error);

        69:
            // Press MESSAGE_CONFIRM_SKIP_PLATE
            result := RaiseMessageBox(Header   := 'Confirm Skip Current Plate',
                                      Message1 := 'Are you sure you want to skip current plate?',
                                      Btn1     := 'GO BACK',
                                      Btn5     := 'CONFIRM',
                                      Severity := TcEventSeverity.Error);

        70:
            // Press MESSAGE_CONFIRM_SKIP_PLATE

            // Note: There's a bit of conflicting text in the original code.

            // We'll unify it below.
            result := RaiseMessageBox(Header   := 'Robot not moving home',
                                      Message1 := 'Press robot is currently in the way of the carriages',
                                      Message2 := 'Retry will double check world zone before moving forward',
                                      Message3 := 'Make sure robot speed isnt too low.',
                                      Btn5     := 'Retry',
                                      Severity := TcEventSeverity.Error);

    ELSE
        // Not Valid Message Number

        // The original code appends the ErrorNumber integer to the message.

        // We'll keep the same logic, but we can store it as a separate or inline string.

        // For demonstration, we directly pass in the integer, though we normally would do

        // a conversion. We'll just label it as an unknown message.
        result := RaiseMessageBox(Header   := 'Not Valid Message Number',
                                  Message1 := CONCAT('UIMessageBox was sent message number: ', UINT_TO_STRING(Robot.Handshake.IN.MessageNumber)),
                                  Message3 := 'Contact Support to update message number.',
                                  Btn1     := 'EXIT MSG',
                                  Severity := TcEventSeverity.Error);
    END_CASE;

    IF result <> 0 THEN
        Robot.Handshake.OUT.MessageSolution    := result;
        Robot.Handshake.OUT.MessageAcknowledge := TRUE;
    END_IF
ELSE
    Robot.Handshake.OUT.MessageSolution    := 0;
    Robot.Handshake.OUT.MessageAcknowledge := FALSE;
END_IF;
END_METHOD

END_FUNCTION_BLOCK

// Machine/EquipmentModules/Info Layer/_FB_EquipmentModule_Info
FUNCTION_BLOCK _FB_EquipmentModule_Info EXTENDS FB_EquipmentModule_SR
VAR
    //Data for recipe
    _Task               : ST_Task;
    TESTrecoveryStepNum : DINT;

END_VAR

METHOD CyclicLogic
VAR_INPUT
END_VAR

VAR
    StepInfo : ST_CSV_Step;
END_VAR
IF NOT _InitComplete THEN
    _InitComplete := Initialize();
    RETURN;
END_IF

_Task.Info.TrussID := _Task.CSV.Steps[1].Details[1].Datas[1];

IF THIS^.CurrentState <> E_PMLState.ePMLState_Execute THEN
    _Task.Info.Active := FALSE;
END_IF

SUPER^.CyclicLogic();
END_METHOD

(*! @summary This method contains code which will execute when this PackML module is in the <b>Aborting</b> state*)
METHOD PROTECTED Aborting

VAR
    result : USINT;
END_VAR
CASE _CurrentMode OF
    E_PMLUnitMode.ePMLUnitMode_Production:

        IF _Task.Info.State = E_TaskState.ACTIVE OR _Task.Info.State = E_TaskState.PENDING THEN
            result := RaiseMessageBox(Header   := CONCAT('Abort Requested:', _Task.Info.StationName),
                                      Message1 := CONCAT('How do you want to abort truss ', UDINT_TO_STRING(_Task.Info.CurrentTaskId)),
                                      Message2 := 'ABORT will scrap the truss',
                                      Message3 := 'MANUAL will stop running the truss but allow you to manually build it.',
                                      Message4 := 'RETRY will stop running the truss and requeue it in SAM',
                                      Message5 := 'REFRESH will discard current data and request New Data from SAM',
                                      Btn2     := 'ABORT',
                                      Btn3     := 'MANUAL',
                                      Btn4     := 'RETRY',
                                      Btn5     := 'REFRESH',
                                      Severity := TcEventSeverity.Error);

            IF result = 2 THEN
                _Task.Info.State           := E_TaskState.ABORT;
                _Task.Info.CurrentTaskStep := 0;
                _Task.StatusUpdate         := TRUE;
                _Task.Info.Active          := FALSE;
            ELSIF result = 3 THEN
                _Task.Info.State           := E_TaskState.MANUAL;
                _Task.Info.CurrentTaskStep := 0;
                _Task.StatusUpdate         := TRUE;
                _Task.Info.Active          := FALSE;
           ELSIF result = 4 THEN
                _Task.Info.State           := E_TaskState.ABORT_RETRY;
                _Task.Info.CurrentTaskStep := 0;
                _Task.StatusUpdate         := TRUE;
                _Task.Info.Active          := FALSE;
            ELSIF result = 5 THEN
                _Task.Info.Active          := FALSE;
                _Task.Info.State           := E_TaskState.IDLE;
                _Task.Info.CurrentTaskStep := 0;
                _Task.StatusUpdate         := TRUE;
                _Task.Info.CurrentTaskId   := 0;
            END_IF

        ELSE
            SUPER^.Aborting();
        END_IF

    E_PMLUnitMode.ePMLUnitMode_Maintenance:
        SUPER^.Aborting();

    E_PMLUnitMode.ePMLUnitMode_Manual:
        SUPER^.Aborting();
END_CASE
END_METHOD

METHOD FindBoardForRecovery : UDINT
VAR_INPUT
    BoardID : DINT;
END_VAR

VAR
    i                     : UDINT;
    RecoveryBoardData     : INT;
    RecoveryPickPlaceData : ST_PickPlace;
END_VAR
FOR i := 1 TO MAX_STEP_COUNT DO
    CASE _Task.CSV.Steps[i].seqName OF
        E_CommandName.BoardInfo:
            RecoveryBoardData := STRING_TO_INT(_Task.CSV.Steps[i].Details[1].Datas[2]);

            IF RecoveryBoardData = BoardID THEN
                FindBoardForRecovery := i;
                EXIT;
            ELSE
                FindBoardForRecovery := 0;
            END_IF

        E_CommandName.Board:
            RecoveryBoardData := STRING_TO_INT(_Task.CSV.Steps[i].Details[1].Datas[5]);

            IF RecoveryBoardData = BoardID THEN
                FindBoardForRecovery := i;
                EXIT;
            ELSE
                FindBoardForRecovery := 0;
            END_IF

        E_CommandName.PickPlace:
            PickPlaceParse(_Task.CSV.Steps[i], RecoveryPickPlaceData);
            RecoveryBoardData := RecoveryPickPlaceData.Number;

            IF RecoveryPickPlaceData.Number = BoardID THEN
                FindBoardForRecovery := i;
                EXIT;
            ELSE
                FindBoardForRecovery := 0;
            END_IF

    ELSE
        FindBoardForRecovery := 0;

    END_CASE
END_FOR
END_METHOD

PROPERTY Task : REFERENCE TO ST_Task;
GET
Task REF= _Task;
END_GET
END_PROPERTY

END_FUNCTION_BLOCK

// Machine/EquipmentModules/SamComm/Helper POUs/FB_FrameFifo
(* Tx/Rx (string data) fifo control function block *)
FUNCTION_BLOCK FB_FrameFifo
VAR_INPUT
    bLog    : BOOL   := FALSE; (* TRUE => Enable log message output, FALSE => Disable *)
    sPrefix : STRING := 'Unknown::'; (* Log message description string (allows the identification of log message source) *)
    putObj  : STRING[25000];
    //	sPut		: T_MaxString 	:= ''; (* String message to add (write) to the fifo *)
END_VAR

VAR_OUTPUT
    bOk    : BOOL; (* TRUE = New entry added or removed succesfully, FALSE = Fifo overflow or fifo empty *)
    getObj : STRING[25000];
    nCount : UDINT := 0; (* Number of fifo entries *)
    cbFree : UDINT := 0; (* Free buffer space *)
END_VAR

VAR
    bReset                         : BOOL := TRUE;
    bAdd, bGet, bRelease, bGetFree : BOOL;
    cbSize                         : UDINT;
    fbBuffer                       : FB_MemRingBufferEx;
    buffer                         : ARRAY[-3..PLCPRJ_BUFFER_SIZE] OF BYTE; (* Internal buffer memory *)
    _Send                          : BOOL;
END_VAR

;

ACTION AddTail:
(* Adds new fifo entry *)
fbBuffer.A_AddTail(pBuffer  := ADR(buffer),
                   cbBuffer := SIZEOF(buffer),
                   pWrite   := ADR(putObj),
                   cbWrite  := SIZEOF(putObj),
                   bOk      => bOk,
                   nCount   => nCount,
                   cbSize   => cbSize,
                   cbFree   => cbFree);

IF bOk THEN
    cbFree := PLCPRJ_BUFFER_SIZE - fbBuffer.cbSize; (* Calculate the free buffer space *)

    IF bLog THEN (* Log message *)
        ADSLOGSTR(ADSLOG_MSGTYPE_HINT OR ADSLOG_MSGTYPE_LOG, CONCAT(sPrefix, '<="%s"'), putObj);
    END_IF
END_IF
END_ACTION

ACTION Clear:
(* Resets fifo = clears all data *)
fbBuffer.A_Reset(pBuffer  := ADR(buffer),
                 cbBuffer := SIZEOF(buffer),
                 bOk      => bOk,
                 nCount   => nCount,
                 cbSize   => cbSize,
                 cbFree   => cbFree);

cbFree := PLCPRJ_BUFFER_SIZE; (* Free buffer size *)
END_ACTION

ACTION RemoveHead:
(* Removes oldest fifo entry *)
fbBuffer.A_GetHead(pBuffer  := ADR(buffer),
                   cbBuffer := SIZEOF(buffer),
                   bOk      => bOk,
                   nCount   => nCount,
                   cbSize   => cbSize,
                   cbFree   => cbFree);

IF bOk THEN
    MEMCPY(ADR(getObj), fbBuffer.pRead, MIN(SIZEOF(getObj), fbBuffer.cbRead));
    cbFree := PLCPRJ_BUFFER_SIZE - fbBuffer.cbSize; (* Calculate the free buffer space *)

    fbBuffer.A_FreeHead(pBuffer  := ADR(buffer),
                        cbBuffer := SIZEOF(buffer),
                        bOk      => bOk,
                        nCount   => nCount,
                        cbSize   => cbSize,
                        cbFree   => cbFree);

    IF fbBuffer.bOk THEN
        ; (* Success *)
    ELSE
        ; (* Buffer empty *)
    END_IF
END_IF
END_ACTION

PROPERTY Send : BOOL
GET
Send := _Send;
END_GET
SET
_Send := Send;
END_SET
END_PROPERTY

END_FUNCTION_BLOCK

// Machine/EquipmentModules/SamComm/Helper POUs/FB_LogFifo
(* Log/debug/error message fifo *)
FUNCTION_BLOCK FB_LogFifo
VAR_INPUT
    bLog    : BOOL   := FALSE; (* TRUE => Enable log message output, FALSE => Disable *)
    sPrefix : STRING := 'Unknown::'; (* Log message description string (allows the identification of log message source) *)

    sMessage : STRING := ''; (* String message to add (write) to the fifo *)
    nErrID   : UDINT  := 0; (* Error code to add (write) to the fifo *)
    hSocket  : T_HSOCKET; (* Socket connection handle *)
END_VAR

VAR_OUTPUT
    bOk    : BOOL; (* TRUE = New entry added or removed succesfully, FALSE = Fifo overflow or fifo empty *)
    sGet   : STRING[1000]; (* String entry removed (read) from fifo *)
    nCount : UDINT := 0; (* Number of fifo entries *)
END_VAR

VAR
    fbBuffer : FB_StringRingBuffer; (* Basic (lower level) string buffer control function block *)
    buffer   : ARRAY[0..PLCPRJ_BUFFER_SIZE] OF BYTE; (* Internal buffer memory *)
    sSource  : STRING[1000];
    sPut     : STRING[1000];
END_VAR

;

ACTION Clear:
(* Clears all fifo entries *)
fbBuffer.A_Reset(pBuffer := ADR(buffer), cbBuffer := SIZEOF(buffer), bOk => bOk, nCount => nCount, getValue => sGet);
END_ACTION

ACTION Error:
(* Adds new fifo entry *)
IF nErrID = 0 THEN
    sSource := '::Error: 0x';
ELSIF (nErrID AND 16#80000000) = 16#80000000 THEN
    IF nErrID = 16#80072746 THEN
        sSource := '::Win32 error (the connection is reset by remote side): 0x';
    ELSE
        sSource := '::Win32 error: 0x';
    END_IF
ELSIF (nErrID AND 16#00008100) = 16#00008100 THEN
    CASE nErrID OF
        PLCPRJ_ERROR_RECEIVE_TIMEOUT:
            sSource := '::PLC sample project receive timeout error: 0x';

        PLCPRJ_ERROR_SENDFIFO_OVERFLOW:
            sSource := '::PLC sample project send fifo overflow error: 0x';

        PLCPRJ_ERROR_RECFIFO_OVERFLOW:
            sSource := '::PLC sample project receive fifo overflow error: 0x';

    ELSE
        sSource := '::Other PLC sample project error: 0x';
    END_CASE
ELSIF (nErrID AND 16#00008000) = 16#00008000 THEN
    sSource := '::Internal TCP/IP Connection Server error: 0x';
ELSE
    sSource := '::TwinCAT System error: 0x';
END_IF

sPut := CONCAT(CONCAT(CONCAT(sPrefix, sMessage), sSource), DWORD_TO_HEXSTR(nErrID AND 16#FFFF, 0, FALSE));

fbBuffer.A_AddTail(pBuffer := ADR(buffer), cbBuffer := SIZEOF(buffer), putValue := sPut, bOk => bOk, nCount => nCount);

IF bOk THEN
    IF bLog THEN (* Log error message *)
        ADSLOGSTR(ADSLOG_MSGTYPE_ERROR OR ADSLOG_MSGTYPE_LOG, '%s', sPut);
    END_IF
END_IF
END_ACTION

ACTION Message:
(* Adds new fifo entry *)
sPut := CONCAT(CONCAT(sPrefix, sMessage), CONCAT('::', HSOCKET_TO_STRING(hSocket)));
fbBuffer.A_AddTail(pBuffer := ADR(buffer), cbBuffer := SIZEOF(buffer), putValue := sPut, bOk => bOk, nCount => nCount);

IF bOk THEN
    IF bLog THEN (* Log information message *)
        ADSLOGSTR(ADSLOG_MSGTYPE_HINT OR ADSLOG_MSGTYPE_LOG, '%s', sPut);
    END_IF
END_IF
END_ACTION

ACTION Remove:
(* Removes oldest fifo entry *)
IF nCount = 0 THEN
    sGet := '';
    bOk  := FALSE;
    RETURN;
END_IF

fbBuffer.A_RemoveHead(pBuffer := ADR(buffer), cbBuffer := SIZEOF(buffer), getValue => sGet, bOk => bOk, nCount => nCount);
END_ACTION

END_FUNCTION_BLOCK

// Machine/EquipmentModules/SamComm/FB_ClientConnection
(* This function block implements simple TCP/IP client protocol. *)
FUNCTION_BLOCK FB_ClientConnection
VAR_IN_OUT
    fbTx  : FB_FrameFifo; (* TX fifo *)
    fbRx  : FB_FrameFifo; (* RX fifo *)
    fbLog : FB_LogFifo; (* Log message fifo *)
END_VAR

VAR_INPUT
    sSrvNetID   : T_AmsNetID := ''; (* TwinCAT TCP/IP server network address *)
    sRemoteHost : T_IPv4Addr := '127.0.0.1'; (* IP address of remote server *)
    nRemotePort : UDINT      := 200; (* Remote server port *)
    bEnable     : BOOL       := FALSE; (* TRUE => Enable/connect, FALSE => Disable/disconnect *)
    tReconnect  : TIME       := T#45s; (* Try to reconnect after this time *)
    bLog        : BOOL       := FALSE; (* TRUE => Enable log message output, FALSE => Disable *)
    sPrefix     : STRING     := 'CLIENT::'; (* Log message description string (allows the identification of log message source) *)
END_VAR

VAR_OUTPUT
    eState : E_SocketConnectionState := eSOCKET_DISCONNECTED; (* TCP/IP connection state *)
END_VAR

VAR
    fbConnect   : FB_ClientServerConnection; (* Create/release TCP/IP connection *)
    fbSend      : FB_SocketSend; (* Send TCP/IP data *)
    fbReceive   : FB_SocketReceive; (* Receive TCP/IP data *)
    nState      : BYTE; (* Global state *)
    bSndBusy    : BOOL; (* Tx state *)
    bRcvBusy    : BOOL; (* Rx state *)
    bDisconnect : BOOL; (* Disconnect flag, if set the socket will be closed *)

    fbPollTimer      : TON; (* Receive poll timer *)
    fbResponseTimer  : TON; (* Response timeout timer *)
    fbReconnectTimer : TON; (* Reconnect timer *)

    cbReceived          : UDINT; (* Count of received data bytes *)
    buffer              : ARRAY[0..PLCPRJ_BUFFER_SIZE] OF BYTE; (* Temp. RX buffer *)
    sRxFrame            : STRING[25000];
    sTxFrame            : STRING[25000];
    i                   : UDINT;
    bAbort              : BOOL;
    nLenOfString        : UDINT; (* String length inclusive the null delimiter *)
    bEndOfString        : BOOL := FALSE;
    posDelim            : UDINT;
    zeroBasedDelimIndex : UDINT;
    nDelimLen           : UDINT;
    fullMsgLen          : UDINT;
    leftover            : UDINT;
END_VAR

CASE nState OF
    0: (* Connect *)
        fbConnect(sSrvNetID   := sSrvNetID,
                  nMode       := SEL(bLog, 0, CONNECT_MODE_ENABLEDBG), (* Enable/disable debug messages? *)
                  sRemoteHost := sRemoteHost,
                  nRemotePort := nRemotePort,
                  bEnable     := bEnable,
                  tReconnect  := tReconnect,
                  eState      => eState);

        IF NOT fbConnect.bBusy THEN
            IF NOT fbConnect.bError THEN
                IF eState = eSOCKET_CONNECTED THEN (* We are connected *)

                    fbTx.Clear(sPrefix := CONCAT(sPrefix, 'FB_FrameFifo(sender)::'), bLog := bLog); (* Clear TX fifo (optional) *)
                    fbRx.Clear(sPrefix := CONCAT(sPrefix, 'FB_FrameFifo(receiver)::'), bLog := bLog); (* Clear RX fifo (optional) *)
                    fbLog.Clear(sPrefix := sPrefix, bLog := bLog); (* Clear log fifo (optional) *)
                    bSndBusy    := FALSE;
                    bRcvBusy    := FALSE;
                    bDisconnect := FALSE;
                    cbReceived  := 0;

                    fbPollTimer(IN := FALSE, PT := T#0S);
                    fbResponseTimer(IN := FALSE, PT := PLCPRJ_RECEIVE_TIMEOUT);
                    fbReconnectTimer(IN := FALSE, PT := tReconnect);

                    fbLog.Message(sMessage := 'Connection established!', hSocket := fbConnect.hSocket);
                    nState := 1;
                END_IF
            ELSE (* Connect error => log error *)
                fbLog.Error(sMessage := 'FB_ClientServerConnection()', nErrID := fbConnect.nErrId);
            END_IF
        END_IF

    1: (* Data exchange state *)
        bDisconnect := NOT bEnable OR bDisconnect; (* User/internal disconnect requested? *)

        IF bDisconnect AND NOT bSndBusy AND NOT bRcvBusy THEN
            bDisconnect := FALSE;
            fbLog.Message(sMessage := 'Closing connection!', hSocket := fbConnect.hSocket);
            nState := 2; (* Disconnect *)
        ELSE

            (* ------------------ Send tx data -------------------------------------- *)
            IF NOT bDisconnect AND NOT bSndBusy THEN
                //                IF fbTx._Send THEN
                fbTx.RemoveHead(getObj => sTxFrame); (* Remove oldest string entry *)

                IF fbTx.bOk THEN (* Success *)
                    fbSend(bExecute := FALSE);
                    fbSend(sSrvNetID := sSrvNetID,
                           hSocket   := fbConnect.hSocket,
                           cbLen     := LEN2(ADR(sTxFrame)), (* Send string inclusive string (null) delimiter! *)
                           pSrc      := ADR(sTxFrame), (* Address of the string variable *)
                           bExecute  := TRUE);

                    bSndBusy := TRUE;
                END_IF

            //                END_IF
            ELSE (* Wait until send not busy *)
                fbSend(bExecute := FALSE);

                IF NOT fbSend.bBusy THEN
                    bSndBusy  := FALSE;
                    fbTx.Send := FALSE;

                    IF fbSend.bError THEN (* Send error => log error and disconnect *)
                        fbLog.Error(sMessage := 'FB_SocketSend()', nErrID := fbSend.nErrId);
                        bDisconnect := TRUE; (* Set flag *)
                    END_IF
                END_IF
            END_IF

            (* ---------------------------------------------------------------------- *)

            (* ---------------------- Get rx data ----------------------------------- *)

            // ----------------- RECEIVE logic updated here ---------------
            IF NOT bDisconnect AND NOT bRcvBusy THEN
                fbPollTimer(IN := TRUE);

                IF fbPollTimer.Q THEN
                    // Enough free room in fbRx & local buffer?
                    IF fbRx.cbFree >= SIZEOF(sRxFrame) THEN
                        fbPollTimer(IN := FALSE, PT := PLCPRJ_RECEIVE_POLLING_TIME);
                        fbReceive(bExecute := FALSE);

                        fbReceive(sSrvNetId := sSrvNetID,
                                  hSocket   := fbConnect.hSocket,
                                  cbLen     := SIZEOF(buffer) - cbReceived,
                                  pDest     := ADR(buffer) + cbReceived,
                                  bExecute  := TRUE);

                        bRcvBusy := TRUE;
                    END_IF
                END_IF

            ELSE
                // Wait until receive is done
                fbReceive(bExecute := FALSE);

                IF NOT fbReceive.bBusy THEN
                    bRcvBusy := FALSE;

                    IF NOT fbReceive.bError THEN

                        IF fbReceive.nRecBytes > 0 THEN
                            // We got fresh bytes. Update how many are in 'buffer'
                            cbReceived := cbReceived + fbReceive.nRecBytes;

                            // Null-terminate the buffer portion to use FIND2

                            // (So we can treat 'buffer' as a normal string for FIND2)
                            //buffer[cbReceived] := 0;

                            // We might get multiple packets in one read,

                            // so keep extracting until no more complete messages.
                            WHILE TRUE DO
                                // Use FIND2 to locate the delimiter in 'buffer'.

                                // This returns 1-based index or 0 if not found.

                                // Adjust the search if your code doesn't allow

                                // direct pointer usage. Usually:

                                //     posDelim := FIND2(ADR(buffer), ADR('>>>endOfPacket__'));

                                // works if 'buffer' is validly null-terminated.
                                posDelim := FIND2(ADR(buffer), ADR('>>>endOfPacket__'));

                                IF posDelim = 0 THEN
                                    // Not found => partial message left in buffer, wait for more
                                    EXIT;
                                END_IF

                                // Because FIND2 is 1-based, convert to zero-based
                                zeroBasedDelimIndex := posDelim - 1;

                                // The delimiter has length 16 = LEN('>>>endOfPacket__')
                                nDelimLen  := 16;
                                fullMsgLen := zeroBasedDelimIndex + nDelimLen;

                                // Check boundary. If it somehow extends beyond cbReceived, break out
                                IF fullMsgLen > cbReceived THEN
                                    // Very unlikely if FIND2 found it, but just to be safe
                                    EXIT;
                                END_IF

                                // Copy that entire packet out to sRxFrame
                                MEMSET(ADR(sRxFrame), 0, SIZEOF(sRxFrame));
                                MEMCPY(ADR(sRxFrame), ADR(buffer), MIN(fullMsgLen, SIZEOF(sRxFrame)));

                                // Push the complete message up to the Rx FIFO
                                fbRx.AddTail(putObj := sRxFrame);

                                IF fbRx.bOk THEN
                                    MEMMOVE(ADR(buffer), ADR(buffer[fullMsgLen]), fullMsgLen); (* Move/shift remaining bytes in buffer *)

                                ELSE
                                    // Overflow in receiving queue
                                    fbLog.Error(sMessage := 'FB_FrameFifo(receiver)', nErrID := PLCPRJ_ERROR_RECFIFO_OVERFLOW);
                                    bDisconnect := TRUE;
                                    RETURN;
                                END_IF

                                // Shift leftover bytes in 'buffer' down
                                leftover := cbReceived - fullMsgLen;

                                //IF leftover > 0 THEN
                                //    MEMMOVE(ADR(buffer), ADR(buffer[fullMsgLen]), leftover);
                                //END_IF

                                cbReceived := leftover;

                                // Loop again if there's another message in the buffer
                            END_WHILE

                            // We received some bytes, so turn off the response timer
                            fbPollTimer(IN := FALSE, PT := T#0S);
                            fbResponseTimer(IN := FALSE);

                        ELSE
                            // No bytes => start/continue the response timeout
                            fbResponseTimer(IN := TRUE);

                            IF fbResponseTimer.Q THEN
                                fbResponseTimer(IN := FALSE);
                                fbLog.Error(sMessage := 'FB_SocketReceive()', nErrID := PLCPRJ_ERROR_RECEIVE_TIMEOUT);
                                bDisconnect := TRUE;
                            END_IF
                        END_IF

                    ELSE
                        // Hard receive error => disconnect
                        fbLog.Error(sMessage := 'FB_SocketReceive()', nErrID := fbReceive.nErrId);
                        bDisconnect := TRUE;
                    END_IF
                END_IF
            END_IF
            // ------------------------------------------------------------
        END_IF

    2: (* Disconnect *)
        fbConnect(bEnable := FALSE, eState => eState);

        IF eState = eSOCKET_DISCONNECTED THEN
            fbReconnectTimer(IN := TRUE); (* Please wait some seconds and then try to connect again *)

            IF fbReconnectTimer.Q THEN
                fbReconnectTimer(IN := FALSE);
                nState := 0;
            END_IF
        END_IF

END_CASE

END_FUNCTION_BLOCK

// Machine/EquipmentModules/SamComm/FB_SamComm
FUNCTION_BLOCK FB_SamComm EXTENDS FB_EquipmentModule_SR
VAR
    // Sub module definitions here

    // List of sub modules

    ipSubModules_Init : ARRAY[1..Parameters_PackML_Base.MAX_NO_OF_SUBMODULES] OF I_PackML_BaseModule := [];

    // Component definitions here

    // List of Components

    ipComponents_Init : ARRAY[1..Parameters_PackML_Base.MAX_NO_OF_COMPONENTS] OF I_ComponentBase := [];

    Line1Empty                : BOOL := FALSE;
    Line2Empty                : BOOL := FALSE;
    InfeedAlternateLine       : BOOL := FALSE;
    InfeedPreviousLineRequest : INT;
END_VAR

VAR
    sSrvNetID : T_AmsNetID := ''; (* TwinCAT TCP/IP server network address *)
    bEnable   : BOOL       := TRUE; (* TRUE => enable client data exchange, FALSE => disable *)
    bLog      : BOOL       := FALSE; (* TRUE => Enable message/error log, FALSE => Disable *)

    fbCloseAll  : FB_SocketCloseAll;
    bInitialize : BOOL := TRUE;

    _Tasks : ARRAY[1..MAX_TASKS] OF ST_TaskREF;

    _OutfeedConveyorStatus_Jig2 : ST_OutfeedConveyorStatus;
    _OutfeedConveyorStatus_Jig3 : ST_OutfeedConveyorStatus;

END_VAR

(* Connection parameters *)

VAR CONSTANT
    //     SERVER_IP : STRING := '192.168.10.100'; (* IP address of the SAM server local at Sawtooth *)
    SERVER_IP   : STRING := '192.168.10.52'; (* IP address of the SAM server *)
    SERVER_PORT : UINT   := 3006; (* Port for SAM server *)
END_VAR

VAR
    eState       : E_SocketConnectionState := eSOCKET_DISCONNECTED; (* TCP/IP connection state *)
    sPrefix      : STRING                  := 'CLIENT::'; (* Log message description string (allows the identification of log message source) *)
    fbConnection : FB_ClientConnection; (* Client data exchange control function block *)
    fbTx         : FB_FrameFifo; (* Tx fifo *)
    fbRx         : FB_FrameFifo; (* Rx fifo *)
    fbLog        : FB_LogFifo; (* Log/debug/error fifo *)

    eStateMachine : E_SAMCommStateMachine := E_SAMCommStateMachine.CREATE_RFI; (* State machine *)
    eStateMachine_PreviousState : E_SAMCommStateMachine; (* State machine *)
    sToServer        : STRING[25000];
    sFromServer      : STRING[25000];
    fbSndTimer       : TON;
    RFT_Index        : INT         := 1;
    sLogMessage      : T_MaxString := '';
    InfeedLineNumber : INT;

    UseLineOneOnly : BOOL := FALSE;

	CurrentMessageUID : STRING[40];
	CurrentMessageCategory : STRING[20];
	
END_VAR

VAR CONSTANT
    PROTOCOL_VERSION     : STRING := 'TRUS.0.1';
    MESSAGE_START        : STRING := 'startOfPacket<<<';
    MESSAGE_END          : STRING := '>>>endOfPacket__';
    HEADER_SPACES        : STRING := '  ';
    MESSAGE_START_LEN    : INT    := 16;
    PROTOCOL_VERSION_OFS : INT    := MESSAGE_START_LEN;
    PROTOCOL_VERSION_LEN : INT    := 8;
    CONTENT_TYPE_OFS     : INT    := PROTOCOL_VERSION_OFS + PROTOCOL_VERSION_LEN;
    CONTENT_TYPE_LEN     : INT    := 8;
    SPACES_ONE_OFS       : INT    := CONTENT_TYPE_OFS + CONTENT_TYPE_LEN;
    SPACES_ONE_LEN       : INT    := 2;
    DATA_LEN_OFS         : INT    := SPACES_ONE_OFS + SPACES_ONE_LEN;
    DATA_LEN_LEN         : INT    := 12;
    SPACES_TWO_OFS       : INT    := DATA_LEN_OFS + DATA_LEN_LEN;
    SPACES_TWO_LEN       : INT    := 2;
    DATA_OFS             : INT    := SPACES_TWO_OFS + SPACES_TWO_LEN;
    MESSAGE_END_LEN      : UDINT  := 16;
    MESSAGE_HEADER_SIZE  : UDINT  := 48;
    MESSAGE_SIZE_MIN     : INT    := 64;
    MESSAGE_DATA_MAX     : UDINT  := (PLCPRJ_BUFFER_SIZE - (MESSAGE_HEADER_SIZE + MESSAGE_END_LEN));
END_VAR

METHOD CyclicLogic
VAR_INPUT
END_VAR
IF NOT _InitComplete THEN
    _InitComplete := Initialize();
    RETURN;
END_IF

SUPER^.CyclicLogic();

(* On PLC reset or program download close all old (opened) connections *)

fbCloseAll(sSrvNetID := sSrvNetID, bExecute := _InitComplete);

IF fbCloseAll.bBusy OR fbCloseAll.bError THEN
    RETURN;
END_IF

//fbClient(sSrvNetId := sSrvNetID, bEnable := bEnable, bLog := bLog);

(*-------------------------- Trigger data exchange -----------------------------------------------*)

fbConnection(sSrvNetID   := sSrvNetID,
             fbRx        := fbRx,
             fbTx        := fbTx,
             fbLog       := fbLog,
             bEnable     := bEnable,
             sRemoteHost := SERVER_IP,
             nRemotePort := SERVER_PORT,
             bLog        := bLog,
             sPrefix     := sPrefix,
             eState      => eState);

IF fbConnection.eState = eSOCKET_CONNECTED THEN (* Connection established *)
    Application();
    //fbApplication( fbTx := fbTx, fbRx := fbRx, fbLog := fbLog );
END_IF
END_METHOD

METHOD CheckForRFT : BOOL
VAR_INPUT
END_VAR

VAR_IN_OUT
    RFT_Task : INT; // Equivalent of Task *out_task
END_VAR

VAR
    i : INT;
END_VAR
// FOR i := 1 TO MAX_TASKS DO
//     IF _Tasks[i].Task.RFT_Requested THEN
//         RFT_Task    := i;
//         CheckForRFT := TRUE;
//         RETURN;
//     END_IF
// END_FOR

FOR i := RFT_Task TO MAX_TASKS DO

    IF _Tasks[i].Task.Info.State <> E_TaskState.INVALID AND _Tasks[i].Task.Info.Active THEN
        IF i > 1 THEN
            IF NOT IsIdleTask(_Tasks[i - 1].Task.Info.State) AND _Tasks[i - 1].Task.Info.CurrentTaskId <> _Tasks[i].Task.Info.CurrentTaskId THEN
                IF IsIdleTask(_Tasks[i].Task.Info.State) THEN
                    fbLog.Message(sMessage := 'Task is idle or completed. Will send RFT after next status...');
                    RFT_Task                     := i; // Update out_task
                    CheckForRFT                  := TRUE;
                    _Tasks[i].Task.RFT_Requested := TRUE;
                    Trace(CONCAT('Task is idle or completed. Will send RFT after next status...: Task # -> ', INT_TO_STRING(RFT_Index)));
                    RETURN;
                END_IF;
            END_IF
        ELSIF i = 1 THEN
            IF IsIdleTask(_Tasks[i].Task.Info.State) THEN
                fbLog.Message(sMessage := 'Task is idle or completed. Will send RFT after next status...');
                RFT_Task                     := i; // Update out_task
                CheckForRFT                  := TRUE;
                _Tasks[i].Task.RFT_Requested := TRUE;
                Trace(CONCAT('Task is idle or completed. Will send RFT after next status...: Task # -> ', INT_TO_STRING(RFT_Index)));
                RETURN;
            END_IF;
        END_IF
    END_IF;
END_FOR;

RFT_Task    := 1;
CheckForRFT := FALSE;
END_METHOD

METHOD CheckForStatusUpdate : BOOL
VAR_INPUT
END_VAR

VAR_IN_OUT
    RFT_Task : INT; // Equivalent of Task *out_task
END_VAR

VAR
    i : INT;
END_VAR
CheckForStatusUpdate := FALSE;
FOR i := RFT_Task TO MAX_TASKS DO
    IF _Tasks[i].Task.Info.State <> E_TaskState.INVALID THEN
        IF _Tasks[i].Task.StatusUpdate THEN
            CheckForStatusUpdate := TRUE;
            EXIT;
        END_IF;
    END_IF;
END_FOR;

FOR i := RFT_Task TO MAX_TASKS DO
    IF CheckForStatusUpdate THEN
        fbLog.Message(sMessage := 'Task has marked status needed, Will send Status before RFT...');
        Trace(CONCAT('Task has marked status needed, Will send Status before RFT...: Task # -> ', INT_TO_STRING(RFT_Index)));
        _Tasks[i].Task.StatusUpdate := FALSE;
    END_IF;
END_FOR;
END_METHOD

METHOD ComposeRequestForInfo : STRING[1000]
VAR_INPUT
END_VAR

VAR
    sPayload          : STRING[1000];
    sTempPayload      : STRING[255];
    sTempPayload2     : STRING[255];
    nPayloadLength    : UDINT;
    nLENofPayloadSize : INT;
    sLENofPayloadSize : STRING(36);
    sRequestMessage   : STRING[1000];
    uuid_str          : STRING(36);
    fbTime            : FB_LocalSystemTime := (bEnable := TRUE);
    currentDateTime   : DATE_AND_TIME;
END_VAR
(* Compose the JSON payload using CONCAT2 *)
fbTime(bEnable := TRUE, dwCycle := 1);
currentDateTime := SYSTEMTIME_TO_DT(fbTime.systemTime);

sPayload := '';

sTempPayload := '{"MessageUuid":"';
CONCAT2(ADR(sPayload), ADR(sTempPayload), ADR(sPayload), SIZEOF(sPayload));
sTempPayload := GenUUID();
CONCAT2(ADR(sPayload), ADR(sTempPayload), ADR(sPayload), SIZEOF(sPayload));
sTempPayload := '","MessageCategory":"RequestForInfo",';
CONCAT2(ADR(sPayload), ADR(sTempPayload), ADR(sPayload), SIZEOF(sPayload));
sTempPayload := '"InResponseToUuid":null,';
CONCAT2(ADR(sPayload), ADR(sTempPayload), ADR(sPayload), SIZEOF(sPayload));
sTempPayload := '"TimeStamp":';
CONCAT2(ADR(sPayload), ADR(sTempPayload), ADR(sPayload), SIZEOF(sPayload));
sTempPayload := DINT_TO_STRING(DT_TO_DINT(currentDateTime));
CONCAT2(ADR(sPayload), ADR(sTempPayload), ADR(sPayload), SIZEOF(sPayload));
sTempPayload := ',"DeviceInfo":{"Name":"AMD PLC","Model":"Beckhoff PLC","Serial":"1234-ABC-12","OSVersion":"9.46","SoftwareVersion":"0.0.1","SoftwareSHA":"abc1234","LogPort":9090,"SecondsSinceBoot":';
CONCAT2(ADR(sPayload), ADR(sTempPayload), ADR(sPayload), SIZEOF(sPayload));
sTempPayload := DWORD_TO_STRING(TIME_TO_DWORD(TIME()));
CONCAT2(ADR(sPayload), ADR(sTempPayload), ADR(sPayload), SIZEOF(sPayload));
sTempPayload := '}}';
CONCAT2(ADR(sPayload), ADR(sTempPayload), ADR(sPayload), SIZEOF(sPayload));

nPayloadLength    := LEN2(ADR(sPayload));
nLENofPayloadSize := LEN(UDINT_TO_STRING(nPayloadLength));
sLENofPayloadSize := UDINT_TO_STRING(nPayloadLength);

(* Construct the full message with headers and footers using CONCAT2 *)
sRequestMessage := '';
CONCAT2(ADR(sRequestMessage), ADR(MESSAGE_START), ADR(sRequestMessage), SIZEOF(sRequestMessage));
CONCAT2(ADR(sRequestMessage), ADR(PROTOCOL_VERSION), ADR(sRequestMessage), SIZEOF(sRequestMessage));
sTempPayload := '    JSON  ';
CONCAT2(ADR(sRequestMessage), ADR(sTempPayload), ADR(sRequestMessage), SIZEOF(sRequestMessage));
sTempPayload := REPLACE('000000000000', sLENofPayloadSize, nLENofPayloadSize, 13 - nLENofPayloadSize);
CONCAT2(ADR(sRequestMessage), ADR(sTempPayload), ADR(sRequestMessage), SIZEOF(sRequestMessage));
sTempPayload := '  ';
CONCAT2(ADR(sRequestMessage), ADR(sTempPayload), ADR(sRequestMessage), SIZEOF(sRequestMessage));
//Add Payload in
CONCAT2(ADR(sRequestMessage), ADR(sPayload), ADR(sRequestMessage), SIZEOF(sRequestMessage));
sTempPayload := '>>>endOfPacket__';
CONCAT2(ADR(sRequestMessage), ADR(sTempPayload), ADR(sRequestMessage), SIZEOF(sRequestMessage));

ComposeRequestForInfo := sRequestMessage;
END_METHOD

METHOD ComposeRFT : STRING[25000]
VAR_INPUT
    index : INT;
END_VAR

VAR
    // Function block instances
    fbJson         : FB_JsonSaxWriter;
    fbJsonDataType : FB_JsonReadWriteDataType;
    fbTime         : FB_LocalSystemTime; // Assuming you have this function block for time

    // Variables
    currentDateTime   : DATE_AND_TIME;
    sPayload          : STRING(5000); // Adjust size as needed
    nPayloadLength    : UDINT;
    nLENofPayloadSize : INT;
    sLENofPayloadSize : STRING(10);
    sRequestMessage   : STRING(5000); // Adjust size as needed
    sTempPayload      : STRING(100);

    // Constants (Assuming these are defined somewhere)
    MESSAGE_START    : STRING := 'startOfPacket<<<';
    PROTOCOL_VERSION : STRING := 'TRUS.0.1    ';
    MESSAGE_END      : STRING := '>>>endOfPacket__';

    // Your StatusMessage structure
    RFTMessage : ST_RFT; // Assuming Message_Type is your structure
    i          : INT;
END_VAR
//Getting the Current Timestamp
fbTime(bEnable := TRUE, dwCycle := 1);
currentDateTime := SYSTEMTIME_TO_DT(fbTime.systemTime);

// Assign values to the root fields
RFTMessage.MessageUuid      := GenUUID();
RFTMessage.MessageCategory  := 'RequestForTask';
CurrentMessageUID := RFTMessage.MessageUuid;
CurrentMessageCategory := RFTMessage.MessageCategory;
RFTMessage.InResponseToUuid := ''; // We'll handle serialization as null
RFTMessage.TimeStamp        := DINT_TO_STRING(DT_TO_DINT(currentDateTime));
RFTMessage.LineNumber       := _tasks[index].Task.Info.LineNumber;
RFTMessage.StationName      := _tasks[index].Task.Info.StationName;
RFTMessage.SubStation       := _tasks[index].Task.Info.SubStation;
//RFTMessage.SubAsyncGroup := tasks[index].SubAsyncGroup;

// Build the JSON payload
fbJson.ResetDocument();
fbJsonDataType.AddJsonValueFromSymbol(fbJson, 'ST_RFT', SIZEOF(RFTMessage), ADR(RFTMessage));

// Copy the JSON document into sPayload
fbJson.CopyDocument(sPayload, SIZEOF(sPayload));

nPayloadLength    := LEN2(ADR(sPayload));
nLENofPayloadSize := LEN(UDINT_TO_STRING(nPayloadLength));
sLENofPayloadSize := UDINT_TO_STRING(nPayloadLength);

(* Construct the full message with headers and footers using CONCAT2 *)
sRequestMessage := '';
CONCAT2(ADR(sRequestMessage), ADR(MESSAGE_START), ADR(sRequestMessage), SIZEOF(sRequestMessage));
CONCAT2(ADR(sRequestMessage), ADR(PROTOCOL_VERSION), ADR(sRequestMessage), SIZEOF(sRequestMessage));
sTempPayload := 'JSON  ';
CONCAT2(ADR(sRequestMessage), ADR(sTempPayload), ADR(sRequestMessage), SIZEOF(sRequestMessage));
sTempPayload := REPLACE('000000000000', sLENofPayloadSize, nLENofPayloadSize, 13 - nLENofPayloadSize);
CONCAT2(ADR(sRequestMessage), ADR(sTempPayload), ADR(sRequestMessage), SIZEOF(sRequestMessage));
sTempPayload := '  ';
CONCAT2(ADR(sRequestMessage), ADR(sTempPayload), ADR(sRequestMessage), SIZEOF(sRequestMessage));
//Add Payload in
CONCAT2(ADR(sRequestMessage), ADR(sPayload), ADR(sRequestMessage), SIZEOF(sRequestMessage));
sTempPayload := '>>>endOfPacket__';
CONCAT2(ADR(sRequestMessage), ADR(sTempPayload), ADR(sRequestMessage), SIZEOF(sRequestMessage));

ComposeRFT := sRequestMessage;
END_METHOD

METHOD ComposeStatus : STRING[25000]
VAR_INPUT
END_VAR

VAR
    // Function block instances
    fbJson         : FB_JsonSaxWriter;
    fbJsonDataType : FB_JsonReadWriteDataType;
    fbTime         : FB_LocalSystemTime; // Assuming you have this function block for time

    // Variables
    currentDateTime   : DATE_AND_TIME;
    sPayload          : STRING(5000); // Adjust size as needed
    nPayloadLength    : UDINT;
    nLENofPayloadSize : INT;
    sLENofPayloadSize : STRING(10);
    sRequestMessage   : STRING(5000); // Adjust size as needed
    sTempPayload      : STRING(100);

    // Constants (Assuming these are defined somewhere)
    MESSAGE_START    : STRING := 'startOfPacket<<<';
    PROTOCOL_VERSION : STRING := 'TRUS.0.1    ';
    MESSAGE_END      : STRING := '>>>endOfPacket__';

    // Your StatusMessage structure
    StatusMessage : ST_Messages; // Assuming Message_Type is your structure
    i             : INT;
END_VAR
//Getting the Current Timestamp
fbTime(bEnable := TRUE, dwCycle := 1);
currentDateTime := SYSTEMTIME_TO_DT(fbTime.systemTime);

// Assign values to the root fields
StatusMessage.MessageUuid     := GenUUID();
StatusMessage.MessageCategory := 'Status';
StatusMessage.TimeStamp       := DINT_TO_STRING(DT_TO_DINT(currentDateTime));

CurrentMessageUID := StatusMessage.MessageUuid;
CurrentMessageCategory := StatusMessage.MessageCategory;

// Assign values to the PLC status removing for now as SAM doesn't do anything with this right now
//StatusMessage.Status.Plc.State := 'SUSPENDED';
//StatusMessage.Status.Plc.Message := 'Infeed starved';

// Assign values to the Tasks array
// Task 1

